// TIA Portal V15.1 export
// export: Created 2026-01-15T16:29:43.8011969Z, ExportSetting WithDefaults, WithReadOnly, DisplayName Totally Integrated Automation Portal, DisplayVersion V15.1 Update 8, DisplayName TIA Portal Openness, DisplayVersion V15.1 Update 8, DisplayName STEP 7 Professional, DisplayVersion V15.1 Update 8, DisplayName WinCC Advanced, DisplayVersion V15.1 Update 8
FUNCTION "7. SAVE_REPORT" : Void   // FC7, LAD
{ S7_Optimized_Access := 'TRUE' }
VERSION : 0.1
// stored: AutoNumber false, CodeModifiedDate 2026-01-15T16:25:53.2342694Z, CompileDate 2026-01-15T16:25:53.2888298Z, CreationDate 2026-01-15T16:22:49.8270549Z, HandleErrorsWithinBlock false, InterfaceModifiedDate 2023-12-15T06:44:57.8941631Z, IsConsistent true, IsIECCheckEnabled false, IsKnowHowProtected false, IsWriteProtected false, LibraryConformanceStatus Warning: The object contains access to global data blocks. Warning: The block contains direct access to inputs, outputs, bit memories, indirect access to the registry or indirect access to external memory areas that are unknown at the time of compilation., ModifiedDate 2026-01-15T16:25:53.2342694Z, ParameterModified 2023-12-15T06:44:57.8941631Z, PLCSimAdvancedSupport false, SetENOAutomatically False, StructureModified 2023-12-15T06:44:57.8941631Z, UDAEnableTagReadback false
   VAR_TEMP   // added for the SCL form of the ladder/FBD networks
      _w1 : Bool;
   END_VAR
BEGIN

REGION Network 1: Lưu dữ liệu Cốt liệu
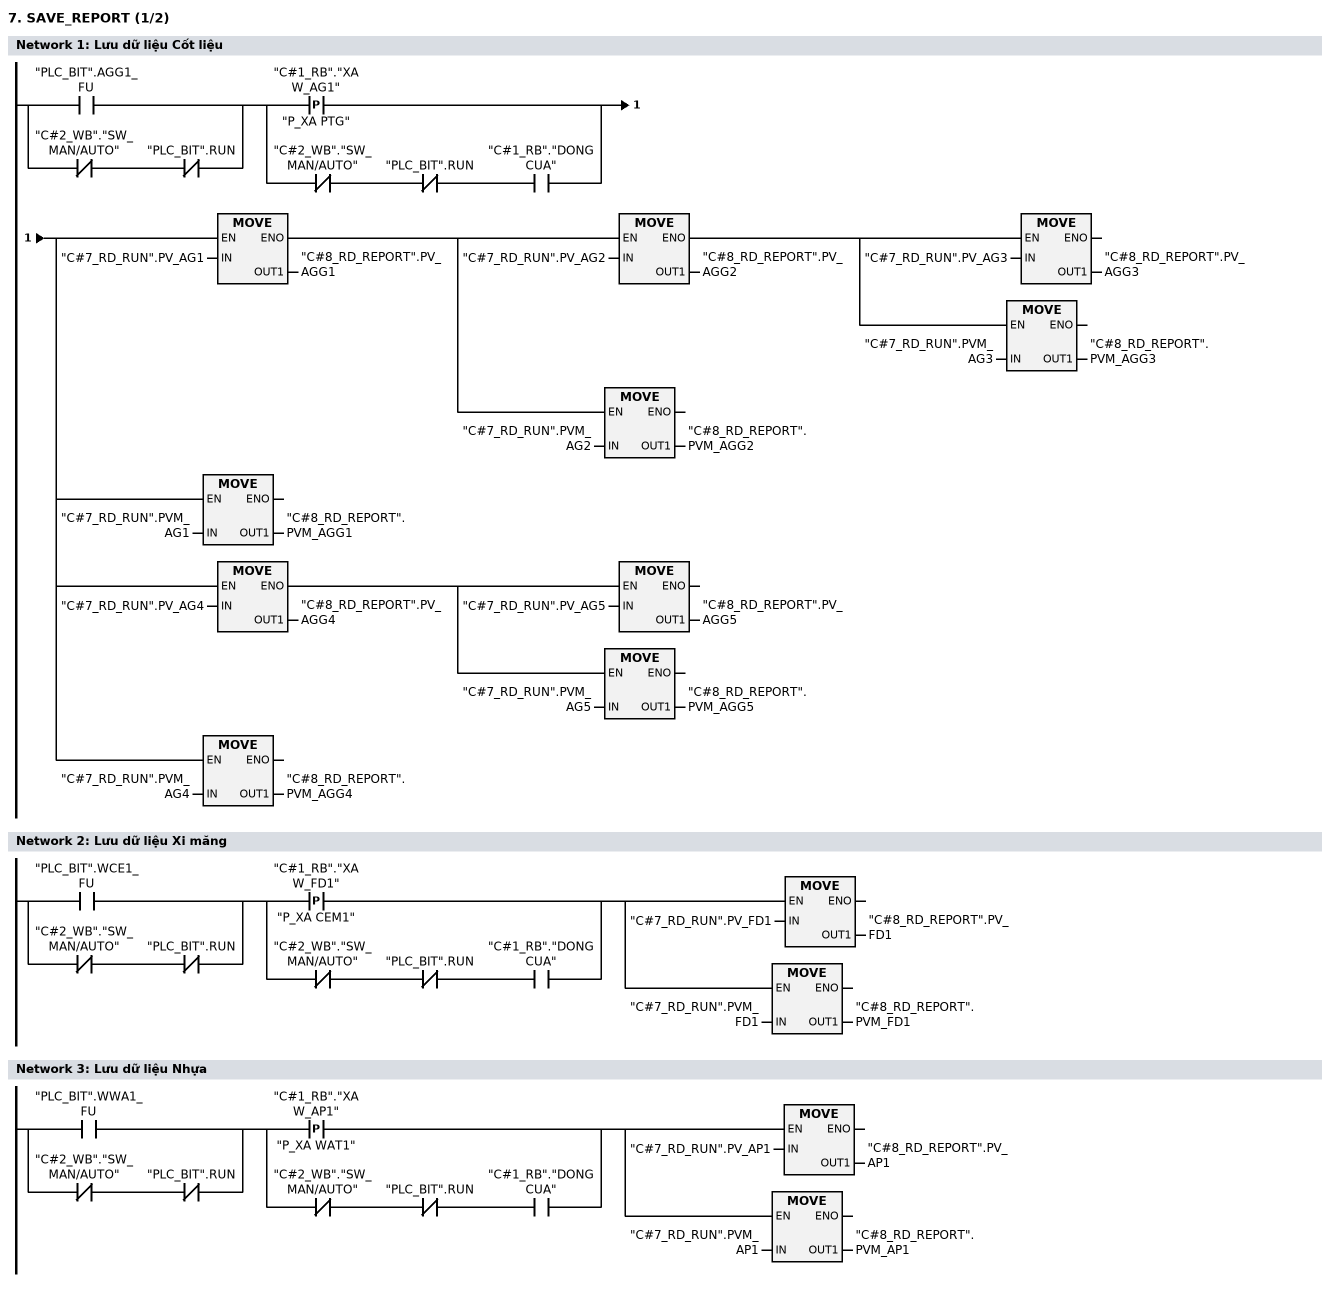
   RUNG wire#powerrail
      Contact( "PLC_BIT".AGG1_FU )
      wire#w1
      P_Contact(operand := "C#1_RB"."XA W_AG1", bit := "P_XA PTG")
      wire#w2
      Move(in := "C#7_RD_RUN".PV_AG1, out1 => "C#8_RD_REPORT".PV_AGG1)
      wire#w3
      Move(in := "C#7_RD_RUN".PV_AG2, out1 => "C#8_RD_REPORT".PV_AGG2)
      wire#w4
      Move(in := "C#7_RD_RUN".PV_AG3, out1 => "C#8_RD_REPORT".PV_AGG3)
   END_RUNG
   RUNG wire#powerrail
      I_Contact( "C#2_WB"."SW_MAN/AUTO" )
      I_Contact( "PLC_BIT".RUN )
   END_RUNG wire#w1
   RUNG wire#w1
      I_Contact( "C#2_WB"."SW_MAN/AUTO" )
      I_Contact( "PLC_BIT".RUN )
      Contact( "C#1_RB"."DONG CUA" )
   END_RUNG wire#w2
   RUNG wire#w4
      Move(in := "C#7_RD_RUN".PVM_AG3, out1 => "C#8_RD_REPORT".PVM_AGG3)
   END_RUNG
   RUNG wire#w3
      Move(in := "C#7_RD_RUN".PVM_AG2, out1 => "C#8_RD_REPORT".PVM_AGG2)
   END_RUNG
   RUNG wire#w2
      Move(in := "C#7_RD_RUN".PVM_AG1, out1 => "C#8_RD_REPORT".PVM_AGG1)
   END_RUNG
   RUNG wire#w2
      Move(in := "C#7_RD_RUN".PV_AG4, out1 => "C#8_RD_REPORT".PV_AGG4)
      wire#w5
      Move(in := "C#7_RD_RUN".PV_AG5, out1 => "C#8_RD_REPORT".PV_AGG5)
   END_RUNG
   RUNG wire#w5
      Move(in := "C#7_RD_RUN".PVM_AG5, out1 => "C#8_RD_REPORT".PVM_AGG5)
   END_RUNG
   RUNG wire#w2
      Move(in := "C#7_RD_RUN".PVM_AG4, out1 => "C#8_RD_REPORT".PVM_AGG4)
   END_RUNG
   // the same network as SCL:
   #_w1 := ("PLC_BIT".AGG1_FU OR (NOT "C#2_WB"."SW_MAN/AUTO" AND NOT "PLC_BIT".RUN)) AND "C#1_RB"."XA W_AG1" AND NOT "P_XA PTG";   // rising edge of "C#1_RB"."XA W_AG1"
   "P_XA PTG" := "C#1_RB"."XA W_AG1";
   IF #_w1 OR (("PLC_BIT".AGG1_FU OR (NOT "C#2_WB"."SW_MAN/AUTO" AND NOT "PLC_BIT".RUN)) AND NOT "C#2_WB"."SW_MAN/AUTO" AND NOT "PLC_BIT".RUN AND "C#1_RB"."DONG CUA") THEN
       "C#8_RD_REPORT".PV_AGG1 := "C#7_RD_RUN".PV_AG1;
       "C#8_RD_REPORT".PV_AGG2 := "C#7_RD_RUN".PV_AG2;
       "C#8_RD_REPORT".PV_AGG3 := "C#7_RD_RUN".PV_AG3;
       "C#8_RD_REPORT".PVM_AGG3 := "C#7_RD_RUN".PVM_AG3;
       "C#8_RD_REPORT".PVM_AGG2 := "C#7_RD_RUN".PVM_AG2;
       "C#8_RD_REPORT".PVM_AGG1 := "C#7_RD_RUN".PVM_AG1;
       "C#8_RD_REPORT".PV_AGG4 := "C#7_RD_RUN".PV_AG4;
       "C#8_RD_REPORT".PV_AGG5 := "C#7_RD_RUN".PV_AG5;
       "C#8_RD_REPORT".PVM_AGG5 := "C#7_RD_RUN".PVM_AG5;
       "C#8_RD_REPORT".PVM_AGG4 := "C#7_RD_RUN".PVM_AG4;
   END_IF;
END_REGION

REGION Network 2: Lưu dữ liệu Xi măng
   RUNG wire#powerrail
      Contact( "PLC_BIT".WCE1_FU )
      wire#w1
      P_Contact(operand := "C#1_RB"."XA W_FD1", bit := "P_XA CEM1")
      wire#w2
      Move(in := "C#7_RD_RUN".PV_FD1, out1 => "C#8_RD_REPORT".PV_FD1)
   END_RUNG
   RUNG wire#powerrail
      I_Contact( "C#2_WB"."SW_MAN/AUTO" )
      I_Contact( "PLC_BIT".RUN )
   END_RUNG wire#w1
   RUNG wire#w1
      I_Contact( "C#2_WB"."SW_MAN/AUTO" )
      I_Contact( "PLC_BIT".RUN )
      Contact( "C#1_RB"."DONG CUA" )
   END_RUNG wire#w2
   RUNG wire#w2
      Move(in := "C#7_RD_RUN".PVM_FD1, out1 => "C#8_RD_REPORT".PVM_FD1)
   END_RUNG
   // the same network as SCL:
   #_w1 := ("PLC_BIT".WCE1_FU OR (NOT "C#2_WB"."SW_MAN/AUTO" AND NOT "PLC_BIT".RUN)) AND "C#1_RB"."XA W_FD1" AND NOT "P_XA CEM1";   // rising edge of "C#1_RB"."XA W_FD1"
   "P_XA CEM1" := "C#1_RB"."XA W_FD1";
   IF #_w1 OR (("PLC_BIT".WCE1_FU OR (NOT "C#2_WB"."SW_MAN/AUTO" AND NOT "PLC_BIT".RUN)) AND NOT "C#2_WB"."SW_MAN/AUTO" AND NOT "PLC_BIT".RUN AND "C#1_RB"."DONG CUA") THEN
       "C#8_RD_REPORT".PV_FD1 := "C#7_RD_RUN".PV_FD1;
       "C#8_RD_REPORT".PVM_FD1 := "C#7_RD_RUN".PVM_FD1;
   END_IF;
END_REGION

REGION Network 3: Lưu dữ liệu Nhựa
   RUNG wire#powerrail
      Contact( "PLC_BIT".WWA1_FU )
      wire#w1
      P_Contact(operand := "C#1_RB"."XA W_AP1", bit := "P_XA WAT1")
      wire#w2
      Move(in := "C#7_RD_RUN".PV_AP1, out1 => "C#8_RD_REPORT".PV_AP1)
   END_RUNG
   RUNG wire#powerrail
      I_Contact( "C#2_WB"."SW_MAN/AUTO" )
      I_Contact( "PLC_BIT".RUN )
   END_RUNG wire#w1
   RUNG wire#w1
      I_Contact( "C#2_WB"."SW_MAN/AUTO" )
      I_Contact( "PLC_BIT".RUN )
      Contact( "C#1_RB"."DONG CUA" )
   END_RUNG wire#w2
   RUNG wire#w2
      Move(in := "C#7_RD_RUN".PVM_AP1, out1 => "C#8_RD_REPORT".PVM_AP1)
   END_RUNG
   // the same network as SCL:
   #_w1 := ("PLC_BIT".WWA1_FU OR (NOT "C#2_WB"."SW_MAN/AUTO" AND NOT "PLC_BIT".RUN)) AND "C#1_RB"."XA W_AP1" AND NOT "P_XA WAT1";   // rising edge of "C#1_RB"."XA W_AP1"
   "P_XA WAT1" := "C#1_RB"."XA W_AP1";
   IF #_w1 OR (("PLC_BIT".WWA1_FU OR (NOT "C#2_WB"."SW_MAN/AUTO" AND NOT "PLC_BIT".RUN)) AND NOT "C#2_WB"."SW_MAN/AUTO" AND NOT "PLC_BIT".RUN AND "C#1_RB"."DONG CUA") THEN
       "C#8_RD_REPORT".PV_AP1 := "C#7_RD_RUN".PV_AP1;
       "C#8_RD_REPORT".PVM_AP1 := "C#7_RD_RUN".PVM_AP1;
   END_IF;
END_REGION

REGION Network 4: Lưu dữ liệu Phụ gia SBS
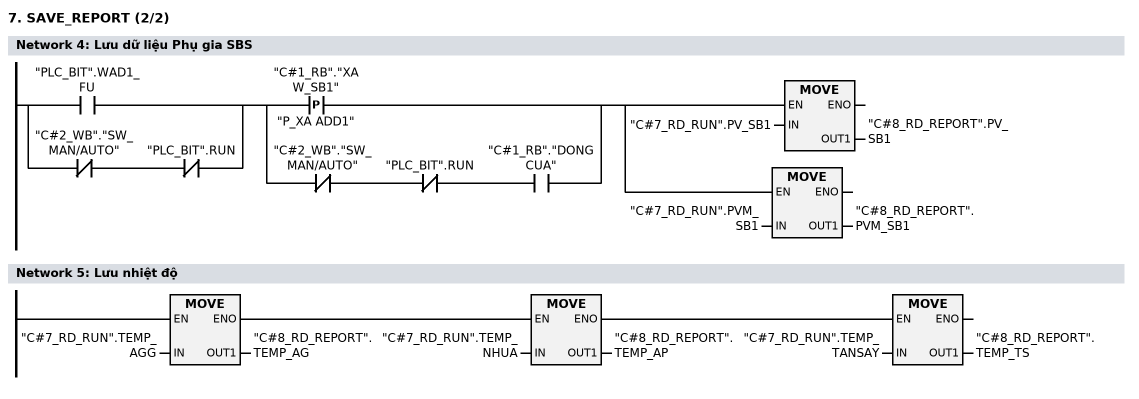
   RUNG wire#powerrail
      Contact( "PLC_BIT".WAD1_FU )
      wire#w1
      P_Contact(operand := "C#1_RB"."XA W_SB1", bit := "P_XA ADD1")
      wire#w2
      Move(in := "C#7_RD_RUN".PV_SB1, out1 => "C#8_RD_REPORT".PV_SB1)
   END_RUNG
   RUNG wire#powerrail
      I_Contact( "C#2_WB"."SW_MAN/AUTO" )
      I_Contact( "PLC_BIT".RUN )
   END_RUNG wire#w1
   RUNG wire#w1
      I_Contact( "C#2_WB"."SW_MAN/AUTO" )
      I_Contact( "PLC_BIT".RUN )
      Contact( "C#1_RB"."DONG CUA" )
   END_RUNG wire#w2
   RUNG wire#w2
      Move(in := "C#7_RD_RUN".PVM_SB1, out1 => "C#8_RD_REPORT".PVM_SB1)
   END_RUNG
   // the same network as SCL:
   #_w1 := ("PLC_BIT".WAD1_FU OR (NOT "C#2_WB"."SW_MAN/AUTO" AND NOT "PLC_BIT".RUN)) AND "C#1_RB"."XA W_SB1" AND NOT "P_XA ADD1";   // rising edge of "C#1_RB"."XA W_SB1"
   "P_XA ADD1" := "C#1_RB"."XA W_SB1";
   IF #_w1 OR (("PLC_BIT".WAD1_FU OR (NOT "C#2_WB"."SW_MAN/AUTO" AND NOT "PLC_BIT".RUN)) AND NOT "C#2_WB"."SW_MAN/AUTO" AND NOT "PLC_BIT".RUN AND "C#1_RB"."DONG CUA") THEN
       "C#8_RD_REPORT".PV_SB1 := "C#7_RD_RUN".PV_SB1;
       "C#8_RD_REPORT".PVM_SB1 := "C#7_RD_RUN".PVM_SB1;
   END_IF;
END_REGION

REGION Network 5: Lưu nhiệt độ
   RUNG wire#powerrail
      Move(in := "C#7_RD_RUN".TEMP_AGG, out1 => "C#8_RD_REPORT".TEMP_AG)
      Move(in := "C#7_RD_RUN".TEMP_NHUA, out1 => "C#8_RD_REPORT".TEMP_AP)
      Move(in := "C#7_RD_RUN".TEMP_TANSAY, out1 => "C#8_RD_REPORT".TEMP_TS)
   END_RUNG
   // the same network as SCL:
   "C#8_RD_REPORT".TEMP_AG := "C#7_RD_RUN".TEMP_AGG;
   "C#8_RD_REPORT".TEMP_AP := "C#7_RD_RUN".TEMP_NHUA;
   "C#8_RD_REPORT".TEMP_TS := "C#7_RD_RUN".TEMP_TANSAY;
END_REGION
END_FUNCTION
